TYPE ST_HW_OutputsTurnTableDTU EXTENDS ST_HW_OutputsTurnTable:

STRUCT
	//Turn table outputs inherits from ST_HW_OutputsTurnTable
	
	//Lift outputs
	Drive_Run_UpDown	: BOOL; // Drive lift up/down	
END_STRUCT
END_TYPE

(* stored: Version 1.1.0.1, ProductVersion 3.1.4024.9
   DUT ST_HW_OutputsTurnTableDTU: Id {bd420360-739b-4d89-ac6e-56d6608834ca} *)
